FUNCTION_BLOCK ExampleDomain_StatusText IMPLEMENTS I_Call
VAR
	_ctx			: REFERENCE TO ExampleDomain_Ctx;
	_fbRec			: Receiver(THIS^);
END_VAR

METHOD Call
VAR_INPUT
	iTag	: Broadcast.Tags.I_Tag;
END_VAR
VAR
	cmp			: TagCmp;
END_VAR
cmp.Set(_ctx.priv.smgr.Current);			

IF cmp.Match(_ctx.state.iExample).IsTrue() THEN
	_ctx.hmi.sStatusText := 'Example State!';
	
	RETURN;
END_IF

IF cmp.IsFalse() THEN
	_ctx.hmi.sStatusText := 'Alarm: Internal Error!';
	
	RETURN;	
END_IF
END_METHOD

//FB_Init is always available implicitly and it is used primarily for initialization.
//The return value is not evaluated. For a specific influence, you can also declare the
//methods explicitly and provide additional code there with the standard initialization
//code. You can evaluate the return value.
METHOD FB_Init: BOOL
VAR_INPUT
    bInitRetains: BOOL; // TRUE: the retain variables are initialized (reset warm / reset cold)
    bInCopyCode: BOOL;  // TRUE: the instance will be copied to the copy code afterward (online change)
	
	ctx			: REFERENCE TO ExampleDomain_Ctx;
END_VAR
_ctx REF= ctx;
ctx.priv.smgr.GetOnChange().Pair(_fbRec);
END_METHOD

METHOD ToDebug : Debug.I_Debug
ToDebug := THIS^;
END_METHOD

END_FUNCTION_BLOCK

(* stored: Version 1.1.0.1
   POU ExampleDomain_StatusText: Id {0417626f-29d8-4c4d-8561-6690e813f16c}, SpecialFunc None
   Method Call: Id {ec843839-0a57-444d-8dab-5f05f06faa31}
   Method FB_init: Id {643b3677-37ca-4b63-845d-ab58a0ac8a8d}
   Method ToDebug: Id {f633fa4d-9995-48df-9ef3-d15fca152da0} *)
